{attribute addProperty BoxType "EK1100-0000-0018"}
{attribute addProperty Id "Beckhoff_EL99xxEK1122Beckhoff_EL99xxEK1122_494C50C5162A_0001_EL9930_0000_0016A_0001_EL9930_0000_0016_8200DBB0364.5"}
{attribute addProperty CRC "3902414817"}
{attribute addProperty SizeInBites "52"}
{attribute addProperty SizeInBytes "6.5"}
TYPE Beckhoff_EL99xx_E89A1FE1 EXTENDS EK1100_179A0949 :
STRUCT
	{attribute addProperty Name "Beckhoff_EL99xxEK1122"}
	Beckhoff_EL99xxEK1122 : Beckhoff_EL99xxEK1122_494C50C5;
	{attribute addProperty Name "A_0001_EL9930_0000_0016"}
	A_0001_EL9930_0000_0016 : A_0001_EL9930_0000_0016_8200DBB0;
END_STRUCT
END_TYPE

(* stored: Version 1.2.0.0, ProductVersion 3.1.4024.9
   DUT Beckhoff_EL99xx_E89A1FE1: Id {bbcf20d6-5f79-4914-a46a-1ca223621ba1} *)
